{attribute addProperty BoxType "EPP9022-0060-0017"}
{attribute addProperty Id "EPM_Inputs_ChannelAT %I*ARRAY[0..1] OF EPM_Inputs_Channel_19E518F4160200WcStateAT %I*WcState_F855686C1620InfoDataAT %I*InfoData_BC63D37F80100"}
{attribute addProperty CRC "2553011981"}
{attribute addProperty SizeInBites "256"}
{attribute addProperty SizeInBytes "32"}
TYPE EPP9022_497E3BE9 :
STRUCT
	{attribute addProperty Name "EPM_Inputs_Channel"}
	EPM_Inputs_Channel : ARRAY[0..1] OF EPM_Inputs_Channel_19E518F4;
	{attribute addProperty Name "WcState"}
	WcState : WcState_F855686C;
	{attribute addProperty Name "InfoData"}
	InfoData : InfoData_BC63D37F;
END_STRUCT
END_TYPE

(* stored: Version 1.2.0.0, ProductVersion 3.1.4024.9
   DUT EPP9022_497E3BE9: Id {c6a732ea-c575-4b0a-9e1c-394d6521b2dd} *)
